TYPE HMI_MAN_General :
STRUCT
	//note: manuals are normally used for controls, not for general
	//PB_MyManualCommand:bool;
END_STRUCT
END_TYPE

(* stored: Version 1.1.0.1
   DUT HMI_MAN_General: Id {42d0f6ab-c743-04e2-2573-e219a6e2b60a} *)
